SYSTEM HVAC2
  (* Version 1.0, 2021-01-14, badger *)
  APPLICATION HVAC2App
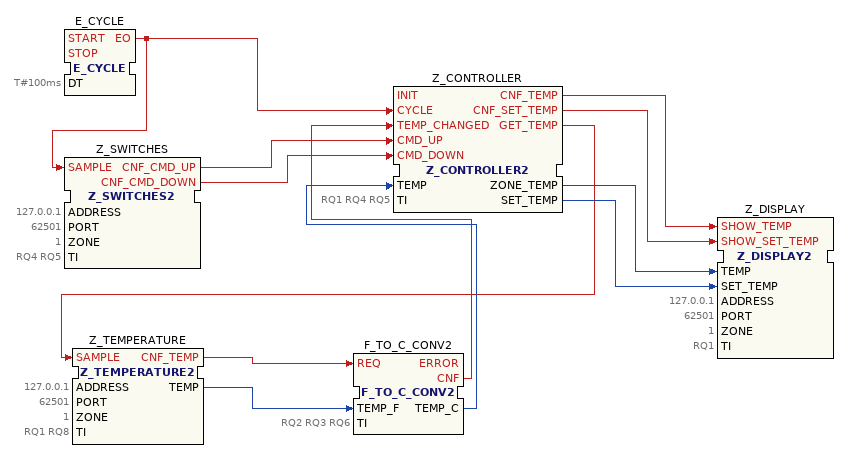
    FBS
      Z_CONTROLLER : Z_CONTROLLER2(TI := RQ1 RQ4 RQ5);
      E_CYCLE : E_CYCLE(DT := T#100ms);
      Z_SWITCHES : Z_SWITCHES2(ADDRESS := 127.0.0.1, PORT := 62501, ZONE := 1, TI := RQ4 RQ5);
      Z_TEMPERATURE : Z_TEMPERATURE2(ADDRESS := 127.0.0.1, PORT := 62501, ZONE := 1, TI := RQ1 RQ8);
      F_TO_C_CONV2 : F_TO_C_CONV2(TI := RQ2 RQ3 RQ6);
      Z_DISPLAY : Z_DISPLAY2(ADDRESS := 127.0.0.1, PORT := 62501, ZONE := 1, TI := RQ1);
    END_FBS
    EVENT_CONNECTIONS
      E_CYCLE.EO TO Z_SWITCHES.SAMPLE;
      E_CYCLE.EO TO Z_CONTROLLER.CYCLE;
      Z_SWITCHES.CNF_CMD_DOWN TO Z_CONTROLLER.CMD_DOWN;
      Z_SWITCHES.CNF_CMD_UP TO Z_CONTROLLER.CMD_UP;
      Z_CONTROLLER.GET_TEMP TO Z_TEMPERATURE.SAMPLE;
      Z_TEMPERATURE.CNF_TEMP TO F_TO_C_CONV2.REQ;
      F_TO_C_CONV2.CNF TO Z_CONTROLLER.TEMP_CHANGED;
      Z_CONTROLLER.CNF_TEMP TO Z_DISPLAY.SHOW_TEMP;
      Z_CONTROLLER.CNF_SET_TEMP TO Z_DISPLAY.SHOW_SET_TEMP;
    END_CONNECTIONS
    DATA_CONNECTIONS
      Z_TEMPERATURE.TEMP TO F_TO_C_CONV2.TEMP_F;
      F_TO_C_CONV2.TEMP_C TO Z_CONTROLLER.TEMP;
      Z_CONTROLLER.ZONE_TEMP TO Z_DISPLAY.TEMP;
      Z_CONTROLLER.SET_TEMP TO Z_DISPLAY.SET_TEMP;
    END_CONNECTIONS
  END_APPLICATION
  DEVICE FORTE_PC : FORTE_PC(MGR_ID := "localhost:61499")
    {SET_ATTRIBUTE(Profile, HOLOBLOC)} (* device profile *)
    RESOURCE EMB_RES : EMB_RES
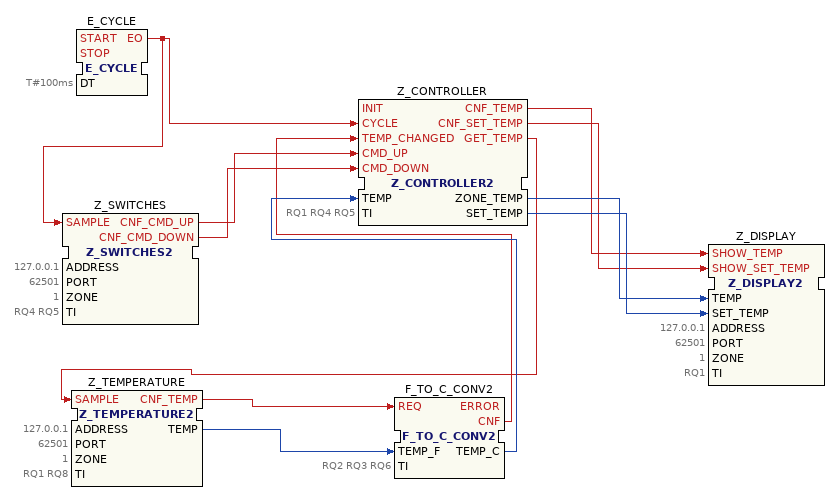
      FBS
        Z_CONTROLLER : Z_CONTROLLER2(TI := RQ1 RQ4 RQ5);
        E_CYCLE : E_CYCLE(DT := T#100ms);
        Z_SWITCHES : Z_SWITCHES2(ADDRESS := 127.0.0.1, PORT := 62501, ZONE := 1, TI := RQ4 RQ5);
        Z_TEMPERATURE : Z_TEMPERATURE2(ADDRESS := 127.0.0.1, PORT := 62501, ZONE := 1, TI := RQ1 RQ8);
        F_TO_C_CONV2 : F_TO_C_CONV2(TI := RQ2 RQ3 RQ6);
        Z_DISPLAY : Z_DISPLAY2(ADDRESS := 127.0.0.1, PORT := 62501, ZONE := 1, TI := RQ1);
      END_FBS
      EVENT_CONNECTIONS
        E_CYCLE.EO TO Z_SWITCHES.SAMPLE;
        E_CYCLE.EO TO Z_CONTROLLER.CYCLE;
        Z_SWITCHES.CNF_CMD_DOWN TO Z_CONTROLLER.CMD_DOWN;
        Z_SWITCHES.CNF_CMD_UP TO Z_CONTROLLER.CMD_UP;
        Z_CONTROLLER.GET_TEMP TO Z_TEMPERATURE.SAMPLE;
        Z_TEMPERATURE.CNF_TEMP TO F_TO_C_CONV2.REQ;
        F_TO_C_CONV2.CNF TO Z_CONTROLLER.TEMP_CHANGED;
        Z_CONTROLLER.CNF_TEMP TO Z_DISPLAY.SHOW_TEMP;
        Z_CONTROLLER.CNF_SET_TEMP TO Z_DISPLAY.SHOW_SET_TEMP;
      END_CONNECTIONS
      DATA_CONNECTIONS
        Z_TEMPERATURE.TEMP TO F_TO_C_CONV2.TEMP_F;
        F_TO_C_CONV2.TEMP_C TO Z_CONTROLLER.TEMP;
        Z_CONTROLLER.ZONE_TEMP TO Z_DISPLAY.TEMP;
        Z_CONTROLLER.SET_TEMP TO Z_DISPLAY.SET_TEMP;
      END_CONNECTIONS
    END_RESOURCE
  END_DEVICE
  MAPPINGS
    HVAC2App.Z_CONTROLLER ON FORTE_PC.EMB_RES.Z_CONTROLLER;
    HVAC2App.E_CYCLE ON FORTE_PC.EMB_RES.E_CYCLE;
    HVAC2App.Z_SWITCHES ON FORTE_PC.EMB_RES.Z_SWITCHES;
    HVAC2App.Z_TEMPERATURE ON FORTE_PC.EMB_RES.Z_TEMPERATURE;
    HVAC2App.F_TO_C_CONV2 ON FORTE_PC.EMB_RES.F_TO_C_CONV2;
    HVAC2App.Z_DISPLAY ON FORTE_PC.EMB_RES.Z_DISPLAY;
  END_MAPPINGS
  SEGMENTS
    Ethernet : Ethernet;
  END_SEGMENTS
  LINKS
    FORTE_PC => Ethernet;
  END_LINKS
END_SYSTEM
